IF k > 9 THEN 
	k := 1;
END_IF;	

IF m > 6 THEN 
	m := 4;
END_IF;

END_PROGRAM

// ---- POUs/csv/P_TextModeWrite_og.TcPOU
(* Writing of CSV file in text mode. None of the field value is containing any non-printing control characters like line feed, carriage return, quotation marks, semicolon... *)
PROGRAM P_TextModeWrite_og
VAR
	bWrite			: BOOL := FALSE;(* Rising edge starts program execution *)
	sNetId			: T_AmsNetId := '';	(* TwinCAT system network address *)
	sFileName		: T_MaxString := 'C:\CSVdata\TextModeGen.csv';(* CSV destination file path and name *)
	sCSVLine		: T_MaxString := '';(* Single CSV text line (row, record), we are using string as record buffer (your are able to see created fields) *)
	sCSVField		: T_MaxString := '';(* Single CSV field value (column, record field) *)
	bBusy			: BOOL;
	bError			: BOOL;
	nErrId			: UDINT;
	nRow	 		: UDINT 	:= 0;(* Row number (record) *)
	nColumn			: UDINT 	:= 0;(* Column number (record field) *)
	hFile			: UINT		:= 0;(* File handle of the source file *)
	step			: DWORD 	:= 0;
	fbFileOpen		: FB_FileOpen;(* Opens file *)
	fbFileClose		: FB_FileClose;(* Closes file *)
	fbFilePuts		: FB_FilePuts;(* Writes one record (line) *)
	fbWriter		: FB_CSVMemBufferWriter;(* Helper function block used to create CSV data bytes (single record line) *)

	database		: ARRAY[0..plc_plc_comm_DB.MAX_CSV_ROWS, 0..plc_plc_comm_DB.MAX_CSV_COLUMNS ] OF STRING(plc_plc_comm_DB.MAX_CSV_FIELD_LENGTH) :=[ (* Source PLC database *)
	'0_0', '0_1', '0_2', '0_3', '0_4', '0_5',
	'1_0', '1_1', '1_2', '1_3', '1_4', '1_5',
	'2_0', '2_1', '2_2', '2_3', '2_4', '2_5',
	'3_0', '3_1', '3_2', '3_3', '3_4', '3_5',
	'4_0', '4_1', '4_2', '4_3', '4_4', '4_5',
	'5_0', '5_1', '5_2', '5_3', '5_4', '5_5'];

END_VAR

CASE step OF
	0:	(* Wait for rising edge at bWrite variable *)
		IF bWrite THEN
			bWrite 	:= FALSE;
			bBusy 	:= TRUE;
			bError	:= FALSE;
			nErrId	:= 0;
			hFile	:= 0;
			nRow	:= 0;
			nColumn	:= 0;
			step 	:= 1;
		END_IF

	1:	(* Open source file *)
		fbFileOpen(  bExecute := FALSE  );
		fbFileOpen( sNetId := sNetId, sPathName := sFileName, nMode := FOPEN_MODEWRITE OR FOPEN_MODETEXT,(* Open file in TEXT mode! *)
					ePath := PATH_GENERIC, bExecute := TRUE );
		step := 2;

	2:(* Wait until open not busy *)
		fbFileOpen( bExecute := FALSE, bError => bError, nErrID => nErrID, hFile => hFile );
		IF NOT fbFileOpen.bBusy THEN
			IF NOT fbFileOpen.bError THEN
				step := 3;
			ELSE(* Error: file not found? *)
				step := 100;
			END_IF
		END_IF

	3:(* Convert one PLC record to CSV format *)
		sCSVLine := '';
		fbWriter.eCmd := eEnumCmd_First;(* Write first field value *)
		IF nRow <= plc_plc_comm_DB.MAX_CSV_ROWS THEN

			FOR nColumn := 0 TO plc_plc_comm_DB.MAX_CSV_COLUMNS BY 1 DO

				sCSVField := STRING_TO_CSVFIELD( database[ nRow, nColumn ], FALSE );(* TODO: Get field value from your application *)

				(* Add new field to the record buffer *)
				fbWriter( 	pBuffer := ADR( sCSVLine ), cbBuffer := SIZEOF( sCSVLine ) - 1, putValue := sCSVField, pValue := 0, cbValue := 0,
							bCRLF := ( nColumn = plc_plc_comm_DB.MAX_CSV_COLUMNS ) );(* bCRLF == TRUE => Write CRLF after the last field value *)
				IF fbWriter.bOk THEN
					fbWriter.eCmd := eEnumCmd_Next;(* Write next field value *)
				ELSE(* Error *)
					step := 100;
					RETURN;
				END_IF

			END_FOR(* FOR nColumn := 0... *)

			(* FB_FilePuts adds allready CR (carriage return) to the written line.
			We have to replace the $R$L characters with $L character to avoid double CR. *)
			IF RIGHT( sCSVLine, 2 ) = '$R$L' THEN
				sCSVLine := REPLACE( sCSVLine, '$L', 2, LEN( sCSVLine ) - 1 );
			END_IF

			nRow := nRow + 1;(* Increment number of created records (rows) *)
			step := 4;(* Write record to the file *)

		ELSE(* All rows written => Close file *)
			step := 10;
		END_IF

	4:	(* Write single text line *)
		fbFilePuts( bExecute := FALSE );
		fbFilePuts( sNetId := sNetId, hFile := hFile, sLine := sCSVLine, bExecute := TRUE );
		step := 5;

	5:(* Wait until write not busy *)
		fbFilePuts( bExecute := FALSE, bError => bError, nErrID => nErrID );
		IF NOT fbFilePuts.bBusy THEN
			IF NOT fbFilePuts.bError THEN
				step := 3;(* Write next record *)
			ELSE(* Error *)
				step := 100;
			END_IF
		END_IF

	10:	(* Close source file *)
		fbFileClose( bExecute := FALSE );
		fbFileClose( sNetId := sNetId, hFile := hFile, bExecute := TRUE );
		step := 11;

	11:(* Wait until close not busy *)
		fbFileClose( bExecute := FALSE, bError => bError, nErrID => nErrID );
		IF ( NOT fbFileClose.bBusy ) THEN
			hFile := 0;
			step := 100;
		END_IF

	100: (* Error or ready step => cleanup *)
		IF ( hFile <> 0 ) THEN
			step := 10; (* Close the source file *)
		ELSE
			bBusy := FALSE;
			step := 0;	(* Ready *)
		END_IF

END_CASE

IF HMI_DB.ChargePB = TRUE THEN 
	bWrite := TRUE;
END_IF

END_PROGRAM

// ---- POUs/Heartbeat.TcPOU
PROGRAM Heartbeat
VAR
	start_TON				: TON;
	start_TON_et 			: TIME;
	reset_TON 				: TON;
	reset_TON_et 			: TIME;
	screen_refresh_pulse 	: BOOL;
	
	pulse_1Hz_Start_TON		: TON;
	pulse_1Hz_Start_PT		: TIME := T#500MS;
	pulse_1Hz_Reset_TON		: TON;
	pulse_1Hz_Reset_PT		: TIME := T#500MS;
	pulse_1Hz				: BOOL;
END_VAR

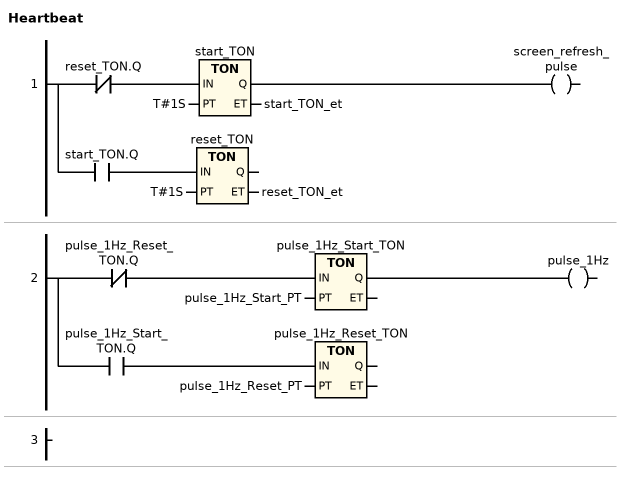
// NETWORK 1
start_TON(IN := NOT reset_TON.Q, PT := T#1S, ET => start_TON_et); // TON
screen_refresh_pulse := start_TON.Q;
reset_TON(IN := start_TON.Q, PT := T#1S, ET => reset_TON_et); // TON

// NETWORK 2
pulse_1Hz_Start_TON(IN := NOT pulse_1Hz_Reset_TON.Q, PT := pulse_1Hz_Start_PT); // TON
pulse_1Hz := pulse_1Hz_Start_TON.Q;
pulse_1Hz_Reset_TON(IN := pulse_1Hz_Start_TON.Q, PT := pulse_1Hz_Reset_PT); // TON

// NETWORK 3

END_PROGRAM

// ---- POUs/HMI.TcPOU
PROGRAM HMI
VAR
	eChargerType : E_ChargerType;
	
	SysCLK					: GETSYSTEMTIME;
	//fileTime				: T_FILETIME;
	LastTimeShot			: STRING;
	ChargeGraphTMR_TON		: TON;
	ChargeGraphTMR_PT		: TIME := ChargeTime_DB.LongestChargeTime_PT + T#10S;
	ChargeGraphTMR_ET		: TIME;
	LongestChargeTIME		: REAL;
	LastTimeShotLog			: BOOL;
	
	i : INT := 1;
	n : INT := 7;

	LastTimeShotTMR_TON		: TON;
	LastTimeShotTMR_PT		: TIME := T#120H;
	LastTimeShotTMR_ET		: TIME;
	LastTimeShotTMR_REAL	: DWORD;
END_VAR

// if clear all faults, reset abort status
IF HMI_DB.ClearFaultPB = TRUE THEN
	Trips_DB.ChargedTimerRunout := FALSE;
	Trips_DB.ChargingTimerRunout := FALSE;
	Trips_DB.DumpTimerRunout := FALSE;
	Trips_DB.ChargerSummaryFault := FALSE;
	Trips_DB.ShortingSystemUnknown := FALSE;
	Trips_DB.AnyEstopPressed := FALSE;
END_IF

IF Trips_DB.ChargedTimerRunout = TRUE OR 
	Trips_DB.ChargingTimerRunout = TRUE //OR 
	//Trips_DB.DumpTimerRunout = TRUE 
	THEN
		Trips_DB.TimerRunOutON := TRUE; 
		ELSE
			Trips_DB.TimerRunOutON := FALSE;
		END_IF


LastTimeShotTMR_TON (IN := TRUE, PT := LastTimeShotTMR_PT, ET => LastTimeShotTMR_ET);

IF (Sequence.eState = E_State.CHARGECOMPLETE) AND HMI_DB.FirePB = TRUE THEN 
	//SysCLK (timeLoDW => fileTime.dwLowDateTime, timeHiDW => fileTime.dwHighDateTime);
	//LastTimeShot := SYSTEMTIME_TO_STRING( FILETIME_TO_SYSTEMTIME( fileTime ) );	
	LastTimeShotTMR_TON (IN := FALSE, PT := LastTimeShotTMR_PT, ET => LastTimeShotTMR_ET);
	HMI_DB.LastTimeShotLog := TRUE;	
	ELSE
		HMI_DB.LastTimeShotLog := FALSE;
END_IF

LastTimeShotTMR_REAL := TIME_TO_DWORD (LastTimeShotTMR_ET)/1000;

IF (Sequence.eState = E_State.CHARGECOMPLETE OR Sequence.eState = E_State.CHARGING) THEN
	ChargeGraphTMR_TON (IN:= TRUE, PT:= ChargeGraphTMR_PT, ET => ChargeGraphTMR_ET);
	ELSE
		ChargeGraphTMR_TON (IN:= FALSE);
END_IF

LongestChargeTIME := TIME_TO_REAL (ChargeGraphTMR_ET)/1000;


IF i > n THEN 
	i := 1;
END_IF

END_PROGRAM

// ---- POUs/LCA_CAL.TcPOU
FUNCTION_BLOCK INTERNAL LCA_CAL
VAR_INPUT
	PSratedV 		: REAL; //kV
	RequiredChargeV	: REAL; //kV
	LoadCapacitance : REAL; //uF
	NumOfCharger	: INT := 1;
	wLCA			: BOOL;
END_VAR
VAR_OUTPUT
	TimeToChargeLoad 	 : REAL;
	RespectedPower		 : REAL;
END_VAR
VAR
	TotalPeakPowerRating : REAL := 9; //kJ/s
	TotalPeakChargeCurrent : REAL;
	AveChargeCurrent 	 : REAL; //A
	LoadStoredEnergy	 : REAL; //J
	Voltage				 : REAL; //
	Volt				 : ARRAY [0..480] OF REAL;
	t					 : ARRAY [0..480] OF REAL;
	deltaT				 : REAL; 
	Icharge				 : ARRAY [0..480] OF REAL;
	Power				 : ARRAY [0..480] OF REAL;
	i : INT := 1;
	j : INT := 1;
	
END_VAR

Volt[0] := 0;
t[0] := 0;
TotalPeakPowerRating := 9 * NumOfCharger;

IF wLCA = FALSE THEN 
	AveChargeCurrent := TotalPeakPowerRating / PSratedV;
	LoadStoredEnergy := 0.5*LoadCapacitance*LREAL_TO_REAL(EXPT(PSratedV, 2));
	//=+(D15*D7/D22)/350
	deltaT := (LoadCapacitance * PSratedV / AveChargeCurrent) / 350; //time step
	//=IF(C35>=(D$9*1000),0,D$22)
	//=+C33+B33*(D$26/1000)/(D$15*0.000001)
	IF Volt[0] >= (RequiredChargeV*1000.5) THEN 
		Icharge[0] := 0;
	ELSE
		Icharge[0] := AveChargeCurrent;
	END_IF
	
	FOR i := 1 TO 480 BY 1 DO 
			
		IF Volt[i] >= (RequiredChargeV*1000.5) THEN 
			Icharge[i] := 0;
		ELSE	
			Icharge[i] := AveChargeCurrent;
		END_IF
		Power[i] := Icharge[i]*Volt[i];
		t[i] := t[i-1]+ deltaT/1000;
		IF Volt[i] >= RequiredChargeV*1000*(0.98) AND Volt[i] <= RequiredChargeV*1000*(1.03) AND Power[i] <> 0 AND Power[i+1] = 0 THEN 
			TimeToChargeLoad := t[i];
			RespectedPower := Power[i];
		END_IF
		Volt[i] := Volt[i-1]+Icharge[i-1]*(deltaT/1000)/(LoadCapacitance*0.000001);
	END_FOR
ELSE//with LCA
	LoadStoredEnergy := 0.5*LoadCapacitance*0.000001*LREAL_TO_REAL(EXPT((RequiredChargeV*1000), 2));
	TotalPeakChargeCurrent := TotalPeakPowerRating*2/PSratedV;
	//IF(C36>=(D$9*1000),0,+IF(C36<500*D$7,D$24,D$24*(0.5+(D$7*1000-C36)/(D$7*1000))))
	deltaT := (LoadCapacitance*PSratedV/TotalPeakChargeCurrent)/350;
				
	IF Volt[i] >= (RequiredChargeV*1000) THEN 
		Icharge[0] := 0;
	ELSIF Volt[i] < (500*PSratedV) THEN
		Icharge[0] := TotalPeakChargeCurrent;
	ELSE
		Icharge[0] := TotalPeakChargeCurrent*(0.5+(PSratedV*1000-Volt[0])/(PSratedV*1000));
	END_IF
	
	FOR i := 1 TO 480 BY 1 DO
			
		IF Volt[i] >= (RequiredChargeV*1000) THEN 
			Icharge[i] := 0;
		ELSE
			IF Volt[i] < (500*PSratedV) THEN
				Icharge[i] := TotalPeakChargeCurrent;
			ELSE
				Icharge[i] := TotalPeakChargeCurrent*(0.5+(PSratedV*1000-Volt[i])/(PSratedV*1000));
			END_IF	
		END_IF
		Volt[i] := Volt[i-1]+Icharge[i-1]*(deltaT/1000)/(LoadCapacitance*0.000001);
		Power[i] := Icharge[i]*Volt[i];
		t[i] := t[i-1]+ deltaT/1000;
		IF Volt[i] >= RequiredChargeV*1000*(0.98) AND Volt[i] <= RequiredChargeV*1000*(1.03) AND Power[i] <> 0 AND Power[i+1] = 0 THEN 
			TimeToChargeLoad := t[i];
			RespectedPower := Power[i];
		END_IF
	END_FOR
END_IF;


IF i > 480 THEN
	i := 1;
END_IF

END_FUNCTION_BLOCK

// ---- POUs/MAIN.TcPOU
PROGRAM MAIN
VAR
END_VAR

Alias();
CAN_comm();
plc_plc_comm();
Permissives();
ChargeTime();
AnalogConversion();
//VoltageMonitor(); - it is done in CAN bus now 
Sequence();
HMI();
//Alarms();
Heartbeat();
RW_CSV();

END_PROGRAM

// ---- POUs/plc_plc_comm.TcPOU
PROGRAM plc_plc_comm
VAR
	ReadfromPLC			: ADSREAD;
	ReadFirePBfromPLC	: ADSREAD;
	WriteStatustoPLC	: ADSWRITE; //P1 PLC need this
	WriteChargTimetoPLC	: ADSWRITE; //P1 PLC need this
	ReadVariableTMR_TON : TON;
END_VAR


ReadVariableTMR_TON(IN := NOT ReadVariableTMR_TON.Q, PT := T#10MS);

//ReadfromPLC (NETID 	:= '192.168.173.60', //p1 pp plc addr - or 5.140.171.248.1.1
ReadfromPLC (NETID 	:= '5.140.171.248.1.1', //p1 pp plc addr - need to be set
			PORT 	:= 851,
			IDXGRP 	:= 16#4020,
			IDXOFFS	:= 16#0,
			LEN		:= SIZEOF(plc_plc_comm_DB.ReadStateFromPLC),
			DESTADDR:= ADR(plc_plc_comm_DB.ReadStateFromPLC), //*MB0
			READ	:= ReadVariableTMR_TON.Q, //high - starts reading
			TMOUT	:= T#2S,
			);
			
ReadFirePBfromPLC (NETID 	:= '5.140.171.248.1.1', //p1 pp plc addr - need to be set
			PORT 	:= 851,
			IDXGRP 	:= 16#4020,
			IDXOFFS	:= 16#008,
			LEN		:= SIZEOF(plc_plc_comm_DB.Button.FirePBPressed),
			DESTADDR:= ADR(plc_plc_comm_DB.Button.FirePBPressed), //*MB8
			READ	:= ReadVariableTMR_TON.Q, //high - starts reading
			TMOUT	:= T#2S,
			);
			
WriteStatustoPLC (NETID   := '5.140.171.248.1.1', //- pfc plc
    		PORT    := 851,
    		IDXGRP  := 16#4020,
    		IDXOFFS := 16#0002,
    		LEN     := SIZEOF(plc_plc_comm_DB.WriteStatetoPLC),
    		SRCADDR := ADR(plc_plc_comm_DB.WriteStatetoPLC), //*MB2
    		WRITE   := ReadVariableTMR_TON.Q,
    		TMOUT   := T#1S,
			);
									
WriteChargTimetoPLC (NETID   := '5.140.171.248.1.1', //- pfc plc
    		PORT    := 851,
    		IDXGRP  := 16#4020,
    		IDXOFFS := 16#0004,
    		LEN     := SIZEOF(plc_plc_comm_DB.ChargeTime),
    		SRCADDR := ADR(plc_plc_comm_DB.ChargeTime), //*MB4
    		WRITE   := ReadVariableTMR_TON.Q,
    		TMOUT   := T#1S,
			);
//read data from the P1_compPP plc and when charge complete (share time count down or use Charge complete status) fire the PFC, 
// wait 2 secs later, close P1_compPP disconnect, does not need feed back signal from this system 
// once disconnect closed, 100ms later, fire woodruff module,
// if no discon closed fb, dump everything <- get dump status from P1_compPP PLC
// this is not needed for M1_CompPP_18M, labview will deal with it

END_PROGRAM

// ---- POUs/Permissives.TcPOU
PROGRAM Permissives
VAR
	
	
END_VAR

//charge relay 
IF (MCP_IO.MagDriver[1].ChargeRelayClose = TRUE (*AND 
	MCP_IO.MagDriver[2].ChargeRelayClose = TRUE AND
	MCP_IO.MagDriver[3].ChargeRelayClose = TRUE AND 
	MCP_IO.MagDriver[4].ChargeRelayClose = TRUE AND 
	MCP_IO.MagDriver[5].ChargeRelayClose = TRUE AND  //uncomment this once we have all 6 racks
	MCP_IO.MagDriver[6].ChargeRelayClose = TRUE*)) OR HMI_DB.AllChargeRelayCloseBP = TRUE
	THEN 
		Permissives_DB.AllChargeRelayClosed := TRUE;
	ELSIF 
		MCP_IO.MagDriver[1].ChargeRelayClose = FALSE (*AND 
		MCP_IO.MagDriver[2].ChargeRelayClose = FALSE AND
		MCP_IO.MagDriver[3].ChargeRelayClose = FALSE AND 
		MCP_IO.MagDriver[4].ChargeRelayClose = FALSE AND 
		MCP_IO.MagDriver[5].ChargeRelayClose = FALSE AND 
		MCP_IO.MagDriver[6].ChargeRelayClose = FALSE*) //uncomment this once we have all 6 racks
	THEN
		Permissives_DB.AllChargeRelayClosed := FALSE;
END_IF;

//dump relay
IF (MCP_IO.MagDriver[1].DumpRelayOpen = TRUE (*AND 
	MCP_IO.MagDriver[2].DumpRelayOpen = TRUE AND
	MCP_IO.MagDriver[3].DumpRelayOpen = TRUE AND
	
	MCP_IO.MagDriver[4].DumpRelayOpen = TRUE AND 
	MCP_IO.MagDriver[5].DumpRelayOpen = TRUE AND //uncomment this once we have all 6 racks
	MCP_IO.MagDriver[6].DumpRelayOpen = TRUE*)) OR HMI_DB.AllDumpRelaysOpenBP = TRUE
	THEN
		Permissives_DB.AllDumpRelayOpen := TRUE;
		ELSIF
			MCP_IO.MagDriver[1].DumpRelayOpen = FALSE (*AND 
			MCP_IO.MagDriver[2].DumpRelayOpen = FALSE AND
			MCP_IO.MagDriver[3].DumpRelayOpen = FALSE AND
			MCP_IO.MagDriver[4].DumpRelayOpen = FALSE AND
			MCP_IO.MagDriver[5].DumpRelayOpen = FALSE AND
			MCP_IO.MagDriver[6].DumpRelayOpen = FALSE *) //uncomment this once we have all 6 racks
		THEN
			Permissives_DB.AllDumpRelayOpen := FALSE;
END_IF;

IF Permissives_DB.AllChargeRelayClosed = TRUE AND 
	Permissives_DB.AllDumpRelayOpen = TRUE   //voltmonitor board has missing packets, so this might be sensitive and might need to bypass
	
	THEN
		Permissives_DB.ReadyToCharge := TRUE;
	ELSE 
		Permissives_DB.ReadyToCharge := FALSE;
END_IF

//charger dc ok
IF MCP_IO.Charger[1].DCOK = TRUE AND 
	MCP_IO.Charger[2].DCOK = TRUE AND 
	MCP_IO.Charger[3].DCOK = TRUE AND
	MCP_IO.Charger[4].DCOK = TRUE AND
	MCP_IO.Charger[5].DCOK = TRUE AND
	MCP_IO.Charger[6].DCOK = TRUE 
	THEN
		Permissives_DB.AllChargerDCOK := TRUE;
	ELSE 
		Permissives_DB.AllChargerDCOK := FALSE;
END_IF
//charger ac ok
IF MCP_IO.Charger[1].ACOK = TRUE AND 
	MCP_IO.Charger[2].ACOK = TRUE AND 
	MCP_IO.Charger[3].ACOK = TRUE AND
	MCP_IO.Charger[4].ACOK = TRUE AND
	MCP_IO.Charger[5].ACOK = TRUE AND
	MCP_IO.Charger[6].ACOK = TRUE 
	THEN
		Permissives_DB.AllChargerACOK := TRUE;
	ELSE 
		Permissives_DB.AllChargerACOK := FALSE;
END_IF

// temperature 
IF MCP_IO.Charger[1].OverTemp = FALSE AND 
	MCP_IO.Charger[2].OverTemp = FALSE AND 
	MCP_IO.Charger[3].OverTemp = FALSE AND
	MCP_IO.Charger[4].OverTemp = FALSE AND
	MCP_IO.Charger[5].OverTemp = FALSE AND
	MCP_IO.Charger[6].OverTemp = FALSE 
	THEN
		Permissives_DB.AllChargerTempOK := TRUE;
	ELSE 
		Permissives_DB.AllChargerTempOK := FALSE;
END_IF

//dump resistor temp 
Permissives_DB.TempThres := HMI_DB.DumpResTempThres;

IF MCP_IO.MagDriver[1].DumpResistorTemp < Permissives_DB.TempThres AND
	MCP_IO.MagDriver[2].DumpResistorTemp < Permissives_DB.TempThres AND
	MCP_IO.MagDriver[3].DumpResistorTemp < Permissives_DB.TempThres AND
	MCP_IO.MagDriver[4].DumpResistorTemp < Permissives_DB.TempThres AND
	MCP_IO.MagDriver[5].DumpResistorTemp < Permissives_DB.TempThres AND
	MCP_IO.MagDriver[6].DumpResistorTemp < Permissives_DB.TempThres
	THEN 
		Permissives_DB.AllDumpResTempOK := TRUE;
		ELSE
			Permissives_DB.AllDumpResTempOK := FALSE;
END_IF



//cap voltage
IF (MCP_IO.MagDriver[1].Cap[1].CapVoltage <= Permissives_DB.CapVoltageThres AND
	MCP_IO.MagDriver[1].Cap[2].CapVoltage <= Permissives_DB.CapVoltageThres AND
	MCP_IO.MagDriver[2].Cap[1].CapVoltage <= Permissives_DB.CapVoltageThres AND
	MCP_IO.MagDriver[2].Cap[2].CapVoltage <= Permissives_DB.CapVoltageThres AND
	MCP_IO.MagDriver[3].Cap[1].CapVoltage <= Permissives_DB.CapVoltageThres AND
	MCP_IO.MagDriver[3].Cap[2].CapVoltage <= Permissives_DB.CapVoltageThres AND
	MCP_IO.MagDriver[4].Cap[1].CapVoltage <= Permissives_DB.CapVoltageThres AND
	MCP_IO.MagDriver[4].Cap[2].CapVoltage <= Permissives_DB.CapVoltageThres AND
	MCP_IO.MagDriver[5].Cap[1].CapVoltage <= Permissives_DB.CapVoltageThres AND
	MCP_IO.MagDriver[5].Cap[2].CapVoltage <= Permissives_DB.CapVoltageThres AND
	MCP_IO.MagDriver[6].Cap[1].CapVoltage <= Permissives_DB.CapVoltageThres AND
	MCP_IO.MagDriver[6].Cap[2].CapVoltage <= Permissives_DB.CapVoltageThres) OR HMI_DB.AllCapsDischargedBP = TRUE 
(*  AND all other module voltage feedback <= 40, might need the -ve end & check for valid data*) 
	THEN
		Permissives_DB.AllCapsDischarged := TRUE;
	ELSE 
		Permissives_DB.AllCapsDischarged := FALSE;
END_IF

IF MCP_IO.MagDriver[1].SCR_ready_to_fire (*AND 
	MCP_IO.MagDriver[2].SCR_ready_to_fire AND 
	MCP_IO.MagDriver[3].SCR_ready_to_fire AND 
	MCP_IO.MagDriver[4].SCR_ready_to_fire AND 
	MCP_IO.MagDriver[5].SCR_ready_to_fire AND 
	MCP_IO.MagDriver[6].SCR_ready_to_fire *)  //uncomment this once we have all 6 racks
	THEN 
		Permissives_DB.AllSCRreadyToFire := TRUE;
		ELSE
			Permissives_DB.AllSCRreadyToFire := FALSE;
END_IF;

IF (//Permissives_DB.AllChargerInhibitON	= TRUE AND 
	Permissives_DB.AllDumpRelayOpen = FALSE AND 
	Permissives_DB.AllCapsDischarged = TRUE) OR HMI_DB.SystemSafeBP = TRUE 
THEN
	(*MCP_IO.Charger[2].voltageFeedback <= 10 AND *)
	Permissives_DB.SystemIsSafe := TRUE;
	ELSE
		Permissives_DB.SystemIsSafe := FALSE;
END_IF
		
IF Permissives_DB.AllCapsDischarged = TRUE THEN 
	MCP_IO.TurnONSystemChargedLED := FALSE; //for status light only
	
END_IF

//MCP_IO.Charger[i].ACOK , DCOK, TEMPOK...

// might or might not beused for the seq
IF MCP_IO.PSU1_DCOK = TRUE AND MCP_IO.Charger[1].ACOK = TRUE  THEN
	Trips_DB.AllDCpsuOK := TRUE;
	ELSE
		Trips_DB.AllDCpsuOK := FALSE;
END_IF

IF MCP_IO.MasterStopPB_NotPressed = FALSE THEN 
	Trips_DB.MasterSTOPPressed := TRUE;
	ELSE
		Trips_DB.MasterSTOPPressed := FALSE;
END_IF

//add logic for e stop
IF MCP_IO.CageEstopCircuitOK = FALSE OR Trips_DB.AnyEstopPressed = FALSE THEN 
	Trips_DB.AnyEstopPressed := TRUE;
END_IF

END_PROGRAM

// ---- POUs/VoltageMonitor.TcPOU
PROGRAM VoltageMonitor
VAR
	i : USINT := 1;
	j : INT := 1;
	k : USINT := 0;
	eVoltFB : E_VoltFB;
	
	m : USINT := 0; //0-18
	n : INT := 0; //
	p : INT := -3;
	q : INT := 3;

	counter : USINT := 0;
	b : ARRAY[0..3] OF BOOL;
	b1 : BOOL;
	b2 : BOOL;
	b3 : BOOL;
	//pause : BOOL;
	//VMBoardWDT_TON : ARRAY[0..24] OF TON;
	//VMBoardWDT_PT	: TIME := T#2S;
	//VMBoardWDT_ET	: TIME;
	//DataNull	: ARRAY[0..24] OF BOOL ;
	//DataNullRebunceTMR_TON : ARRAY[0..24] OF TON;
	//DataNullRebounce_PT	: TIME := T#800MS;
	//DataNullRebounce	: ARRAY[0..24] OF BOOL ;
	VMB1 : ARRAY[0..17] OF VoltTranBd;
	VMB2 : ARRAY[0..17] OF VoltTranBd;
END_VAR

//2 voltage tran borad per module, total of 36 channels for M1 
//volt monitor board 1 - trans board 0
FOR m := 0 TO 17 BY 1 DO 
	VMB1[m] ( CapRaw := LCP1_IO.VMB.VTB[m].CapRaw );		
	LCP1_IO.VMB.VTB[m].BateryLow 						:= VMB1[m].BatteryLow;
	LCP1_IO.VMB.VTB[m].VoltageReading_raw				:= VMB1[m].VoltageReading_raw;
	LCP1_IO.VMB.VTB[m].DataNull							:= VMB1[m].DataNull; 
	LCP1_IO.VMB.VTB[m].LossVoltTransBoard				:= VMB1[m].LossVoltMonitorBoard;			
	
	VMB2[m] ( CapRaw := LCP2_IO.VMB.VTB[m].CapRaw );		
	LCP2_IO.VMB.VTB[m].BateryLow 						:= VMB2[m].BatteryLow;
	LCP2_IO.VMB.VTB[m].VoltageReading_raw				:= VMB2[m].VoltageReading_raw;
	LCP2_IO.VMB.VTB[m].DataNull							:= VMB2[m].DataNull; 
	LCP2_IO.VMB.VTB[m].LossVoltTransBoard				:= VMB2[m].LossVoltMonitorBoard;
END_FOR

//status - add VM.VTB to alarms.
(*
LCP1_IO.Segment[1].Module[1].VTB[1].BateryLow			:= LCP1_IO.VMB.VTB[0].BateryLow;
LCP1_IO.Segment[1].Module[1].VTB[1].DataNull 			:= LCP1_IO.VMB.VTB[0].DataNull;
LCP1_IO.Segment[1].Module[1].VTB[1].LossVoltTransBoard 	:= LCP1_IO.VMB.VTB[0].LossVoltTransBoard;
LCP1_IO.Segment[1].Module[1].VTB[2].BateryLow			:= LCP1_IO.VMB.VTB[1].BateryLow;
LCP1_IO.Segment[1].Module[1].VTB[2].DataNull			:= LCP1_IO.VMB.VTB[1].DataNull;
LCP1_IO.Segment[1].Module[1].VTB[2].LossVoltTransBoard	:= LCP1_IO.VMB.VTB[1].LossVoltTransBoard;

LCP1_IO.Segment[1].Module[2].VTB[1].BateryLow			:= LCP1_IO.VMB.VTB[2].BateryLow;
LCP1_IO.Segment[1].Module[2].VTB[1].DataNull			:= LCP1_IO.VMB.VTB[2].DataNull;
LCP1_IO.Segment[1].Module[2].VTB[1].LossVoltTransBoard	:= LCP1_IO.VMB.VTB[2].LossVoltTransBoard;
LCP1_IO.Segment[1].Module[2].VTB[2].BateryLow			:= LCP1_IO.VMB.VTB[3].BateryLow;
LCP1_IO.Segment[1].Module[2].VTB[2].DataNull			:= LCP1_IO.VMB.VTB[3].DataNull;
LCP1_IO.Segment[1].Module[2].VTB[2].LossVoltTransBoard	:= LCP1_IO.VMB.VTB[3].LossVoltTransBoard;

LCP1_IO.Segment[1].Module[3].VTB[1].BateryLow			:= LCP1_IO.VMB.VTB[4].BateryLow;
LCP1_IO.Segment[1].Module[3].VTB[1].DataNull			:= LCP1_IO.VMB.VTB[4].DataNull;
LCP1_IO.Segment[1].Module[3].VTB[1].LossVoltTransBoard	:= LCP1_IO.VMB.VTB[4].LossVoltTransBoard;
LCP1_IO.Segment[1].Module[3].VTB[2].BateryLow			:= LCP1_IO.VMB.VTB[5].BateryLow;
LCP1_IO.Segment[1].Module[3].VTB[2].DataNull			:= LCP1_IO.VMB.VTB[5].DataNull;
LCP1_IO.Segment[1].Module[3].VTB[2].LossVoltTransBoard	:= LCP1_IO.VMB.VTB[5].LossVoltTransBoard;

LCP1_IO.Segment[2].Module[4].VTB[1].BateryLow			:= LCP1_IO.VMB.VTB[6].BateryLow;
LCP1_IO.Segment[2].Module[4].VTB[1].DataNull			:= LCP1_IO.VMB.VTB[6].DataNull;
LCP1_IO.Segment[2].Module[4].VTB[1].LossVoltTransBoard	:= LCP1_IO.VMB.VTB[6].LossVoltTransBoard;
LCP1_IO.Segment[2].Module[4].VTB[2].BateryLow			:= LCP1_IO.VMB.VTB[7].BateryLow;
LCP1_IO.Segment[2].Module[4].VTB[2].DataNull			:= LCP1_IO.VMB.VTB[7].DataNull;
LCP1_IO.Segment[2].Module[4].VTB[2].LossVoltTransBoard	:= LCP1_IO.VMB.VTB[7].LossVoltTransBoard;

LCP1_IO.Segment[2].Module[5].VTB[1].BateryLow			:= LCP1_IO.VMB.VTB[8].BateryLow;
LCP1_IO.Segment[2].Module[5].VTB[1].DataNull			:= LCP1_IO.VMB.VTB[8].DataNull;
LCP1_IO.Segment[2].Module[5].VTB[1].LossVoltTransBoard	:= LCP1_IO.VMB.VTB[8].LossVoltTransBoard;
LCP1_IO.Segment[2].Module[5].VTB[2].BateryLow			:= LCP1_IO.VMB.VTB[9].BateryLow;
LCP1_IO.Segment[2].Module[5].VTB[2].DataNull			:= LCP1_IO.VMB.VTB[9].DataNull;
LCP1_IO.Segment[2].Module[5].VTB[2].LossVoltTransBoard	:= LCP1_IO.VMB.VTB[9].LossVoltTransBoard;
*)
//FOR i := 1 TO 3 BY 1 DO //segment 1 - 3
(*	IF i = 1 THEN 
		IF p > 0 THEN
			p := -3;
		END_IF 
		p := p + 1;
		j := p + q;	
		FOR k := 1 TO 2 BY 1 DO 		 
			//n vtb 0-17
			n := k + j + p; //
			LCP1_IO.Segment[i].Module[j].VoltageFeedback_raw[k] := LCP1_IO.VMB.VTB[n].VoltageReading_raw;
		END_FOR
	END_IF;
	*)
//END_FOR
(*
CASE eVoltFB OF
	E_VoltFB.seg1:
		i := 1;
		FOR j := 1 TO	3 BY 1 DO //module 1 -9			
			IF p > 0 THEN
				p := -3;
			END_IF 
			p := p + 1;
			j := p + q;	

			FOR k := 1 TO 2 BY 1 DO 		 
				//n vtb 0-17
				n := k + j + p; //
				LCP1_IO.Segment[i].Module[j].VoltageFeedback_raw[k] := LCP1_IO.VMB.VTB[n].VoltageReading_raw;
			END_FOR
			i := i +1;
			eVoltFB := E_VoltFB.seg2;
		END_FOR	
	E_VoltFB.seg2:
		IF p > 3 THEN
			p := 0;
		END_IF 
		p := p + 1;
		j := p + q;	

		FOR k := 1 TO 2 BY 1 DO 		 
				//n vtb 0-17
				n := k + j + p; //
				LCP1_IO.Segment[i].Module[j].VoltageFeedback_raw[k] := LCP1_IO.VMB.VTB[n].VoltageReading_raw;
		END_FOR
		i := i + 1;
		eVoltFB := E_VoltFB.seg3;
	E_VoltFB.seg3:
			IF p > 6 THEN
				p := 3;
			END_IF 
			p := p + 1;
			j := p + q;	

			FOR k := 1 TO 2 BY 1 DO 		 
				//n vtb 0-17
				n := k + j + p; //
				LCP1_IO.Segment[i].Module[j].VoltageFeedback_raw[k] := LCP1_IO.VMB.VTB[n].VoltageReading_raw;
			END_FOR
			i := i + 1;
			eVoltFB := E_VoltFB.seg3;
END_CASE
*)

LCP1_IO.Segment[1].Module[1].VoltageFeedback_raw[1] := LCP1_IO.VMB.VTB[0].VoltageReading_raw;
LCP1_IO.Segment[1].Module[1].VoltageFeedback_raw[2] := LCP1_IO.VMB.VTB[1].VoltageReading_raw;
LCP1_IO.Segment[1].Module[2].VoltageFeedback_raw[1] := LCP1_IO.VMB.VTB[2].VoltageReading_raw;
LCP1_IO.Segment[1].Module[2].VoltageFeedback_raw[2] := LCP1_IO.VMB.VTB[3].VoltageReading_raw;
LCP1_IO.Segment[1].Module[3].VoltageFeedback_raw[1] := LCP1_IO.VMB.VTB[4].VoltageReading_raw;
LCP1_IO.Segment[1].Module[3].VoltageFeedback_raw[2] := LCP1_IO.VMB.VTB[5].VoltageReading_raw;
LCP1_IO.Segment[2].Module[4].VoltageFeedback_raw[1] := LCP1_IO.VMB.VTB[6].VoltageReading_raw;
LCP1_IO.Segment[2].Module[4].VoltageFeedback_raw[2] := LCP1_IO.VMB.VTB[7].VoltageReading_raw;
LCP1_IO.Segment[2].Module[5].VoltageFeedback_raw[1] := LCP1_IO.VMB.VTB[8].VoltageReading_raw;
LCP1_IO.Segment[2].Module[5].VoltageFeedback_raw[2] := LCP1_IO.VMB.VTB[9].VoltageReading_raw;
LCP1_IO.Segment[2].Module[6].VoltageFeedback_raw[1] := LCP1_IO.VMB.VTB[10].VoltageReading_raw;
LCP1_IO.Segment[2].Module[6].VoltageFeedback_raw[2] := LCP1_IO.VMB.VTB[11].VoltageReading_raw;
LCP1_IO.Segment[3].Module[7].VoltageFeedback_raw[1] := LCP1_IO.VMB.VTB[12].VoltageReading_raw;
LCP1_IO.Segment[3].Module[7].VoltageFeedback_raw[2] := LCP1_IO.VMB.VTB[13].VoltageReading_raw;
LCP1_IO.Segment[3].Module[8].VoltageFeedback_raw[1] := LCP1_IO.VMB.VTB[14].VoltageReading_raw;
LCP1_IO.Segment[3].Module[8].VoltageFeedback_raw[2] := LCP1_IO.VMB.VTB[15].VoltageReading_raw;
LCP1_IO.Segment[3].Module[9].VoltageFeedback_raw[1] := LCP1_IO.VMB.VTB[16].VoltageReading_raw;
LCP1_IO.Segment[3].Module[9].VoltageFeedback_raw[2] := LCP1_IO.VMB.VTB[17].VoltageReading_raw;

LCP2_IO.Segment[4].Module[1].VoltageFeedback_raw[1] := LCP2_IO.VMB.VTB[0].VoltageReading_raw;
LCP2_IO.Segment[4].Module[1].VoltageFeedback_raw[2] := LCP2_IO.VMB.VTB[1].VoltageReading_raw;
LCP2_IO.Segment[4].Module[2].VoltageFeedback_raw[1] := LCP2_IO.VMB.VTB[2].VoltageReading_raw;
LCP2_IO.Segment[4].Module[2].VoltageFeedback_raw[2] := LCP2_IO.VMB.VTB[3].VoltageReading_raw;
LCP2_IO.Segment[4].Module[3].VoltageFeedback_raw[1] := LCP2_IO.VMB.VTB[4].VoltageReading_raw;
LCP2_IO.Segment[4].Module[3].VoltageFeedback_raw[2] := LCP2_IO.VMB.VTB[5].VoltageReading_raw;
LCP2_IO.Segment[5].Module[4].VoltageFeedback_raw[1] := LCP2_IO.VMB.VTB[6].VoltageReading_raw;
LCP2_IO.Segment[5].Module[4].VoltageFeedback_raw[2] := LCP2_IO.VMB.VTB[7].VoltageReading_raw;
LCP2_IO.Segment[5].Module[5].VoltageFeedback_raw[1] := LCP2_IO.VMB.VTB[8].VoltageReading_raw;
LCP2_IO.Segment[5].Module[5].VoltageFeedback_raw[2] := LCP2_IO.VMB.VTB[9].VoltageReading_raw;
LCP2_IO.Segment[5].Module[6].VoltageFeedback_raw[1] := LCP2_IO.VMB.VTB[10].VoltageReading_raw;
LCP2_IO.Segment[5].Module[6].VoltageFeedback_raw[2] := LCP2_IO.VMB.VTB[11].VoltageReading_raw;
LCP2_IO.Segment[6].Module[7].VoltageFeedback_raw[1] := LCP2_IO.VMB.VTB[12].VoltageReading_raw;
LCP2_IO.Segment[6].Module[7].VoltageFeedback_raw[2] := LCP2_IO.VMB.VTB[13].VoltageReading_raw;
LCP2_IO.Segment[6].Module[8].VoltageFeedback_raw[1] := LCP2_IO.VMB.VTB[14].VoltageReading_raw;
LCP2_IO.Segment[6].Module[8].VoltageFeedback_raw[2] := LCP2_IO.VMB.VTB[15].VoltageReading_raw;
LCP2_IO.Segment[6].Module[9].VoltageFeedback_raw[1] := LCP2_IO.VMB.VTB[16].VoltageReading_raw;
LCP2_IO.Segment[6].Module[9].VoltageFeedback_raw[2] := LCP2_IO.VMB.VTB[17].VoltageReading_raw;

//add shaft ramp stuff here

IF i > 3 THEN 
	i := 1;
END_IF

IF j > 9 THEN 
	j := 1;
END_IF

IF k > 2 THEN 
	k := 1;
END_IF

IF m > 17 THEN
	m := 0;
END_IF


IF p >= 7 THEN
	p := -3;
END_IF

END_PROGRAM

// ---- POUs/VoltTranBd.TcPOU
FUNCTION_BLOCK VoltTranBd
VAR_INPUT
	CapRaw : UINT;
END_VAR
VAR_OUTPUT
	BatteryLow  		: BOOL;
	VoltageReading		: INT; //custom board
	VoltageReading_raw	: INT;
	DataNull			: BOOL;
	LossVoltMonitorBoard : BOOL := 0;
END_VAR
VAR
	VMBoardWDT_TON :  TON;
	VMBoardWDT_ET	: TIME;
	DataNullRebunceTMR_TON :  TON;
	DataNullRebounce	: BOOL;
	VMBoardWDT_PT		: TIME := T#2S;
	DataNullRebounce_PT	: TIME := T#800MS;
	
END_VAR


	IF CapRaw <> 0 THEN
		VoltageReading_raw.0 := CapRaw.2;
		VoltageReading_raw.1 := CapRaw.3;
		VoltageReading_raw.2 := CapRaw.4;
		VoltageReading_raw.3 := CapRaw.5;
	
		VoltageReading_raw.4 := CapRaw.6;
		VoltageReading_raw.5 := CapRaw.7;
		VoltageReading_raw.6 := CapRaw.8;
		VoltageReading_raw.7 := CapRaw.9;
	
		VoltageReading_raw.8 := CapRaw.10;
		VoltageReading_raw.9 := CapRaw.11;
	
		VoltageReading_raw.10 := 0;//CapRaw.14;
		VoltageReading_raw.11 := 0;//CapRaw.15;
		VoltageReading_raw.12 := 0;//CapRaw.12;
		VoltageReading_raw.13 := 0;//CapRaw.13;
		VoltageReading_raw.14 := 0; //CapRaw.14;
	
		VoltageReading_raw.15 := 0;//VoltMonitor_DB.CapRaw.4;
		
		VMBoardWDT_TON (IN := FALSE);
		ELSE
			VMBoardWDT_TON (IN := TRUE, PT := VMBoardWDT_PT, ET => VMBoardWDT_ET);
			//VoltMonitor_DB.CapRaw_DummySnap[k] := 0;
	END_IF
	
	
	IF VMBoardWDT_TON.Q THEN 
		DataNull := TRUE; 
		LossVoltMonitorBoard := TRUE;
	END_IF
	
	IF DataNull = TRUE THEN
		VoltageReading_raw := ULINT_TO_INT(NULL);
	END_IF
	
	IF LossVoltMonitorBoard = TRUE THEN
		DataNullRebunceTMR_TON( IN := TRUE, PT := DataNullRebounce_PT);
	END_IF

	IF DataNullRebunceTMR_TON.Q = TRUE THEN
		DataNull := FALSE;
		DataNullRebunceTMR_TON( IN := FALSE);
	END_IF
	

	IF DataNull = TRUE THEN
		VoltageReading_raw := ULINT_TO_INT(NULL);
	END_IF;

END_FUNCTION_BLOCK
